(*
Specifies the anti-windup strategy used by :itf:`FB_Integrator`.
*)
{attribute 'qualified_only'}
{attribute 'strict'}
{attribute 'to_string'}
TYPE E_AntiWindupMethod :
(
	// Halts integration when the output is saturated.
	Clamping        := 0, 
	// Feeds back the saturation error to unwind the integrator gradually. 
	// Recommended for slow systems with significant lag
	BackCalculation := 1
)BYTE;
END_TYPE

(* stored: Version 1.1.0.1, ProductVersion 3.1.4024.15
   EnumerationTextList E_AntiWindupMethod: Id {58a5dd66-d53c-4f34-bd90-758e7f6a7e06} *)
